# EPICS substitutions: ek9000App/Db/EL1098.substitutions
file EL1098.template
{ 	pattern
	{
		TERMINAL,

	}
	{
	}
}
